// TIA Portal V16 export
// export: Created 2024-06-17T16:39:12.649221Z, ExportSetting None, DisplayName Totally Integrated Automation Portal, DisplayVersion V16, DisplayName TIA Portal Version Control Interface, DisplayVersion V16, DisplayName TIA Portal Openness, DisplayVersion V16, DisplayName STEP 7 Professional, DisplayVersion V16, DisplayName STEP 7 Safety, DisplayVersion V16, DisplayName WinCC Advanced, DisplayVersion V16
FUNCTION_BLOCK "0105_FB Robô ABB"   // FB105, LAD
TITLE = Assinatura
{ S7_Optimized_Access := 'FALSE' }
AUTHOR : Axis_Solutions
// Autor           : Pedro Mello
// E-mail         : pedro.mello@axissolutions.com.br
// Empresa    : Axis Solutions
// Site             : www.axissolutions.com.br
//                     
// Data de criação : 11.06.2024
// Função                : Gestão de robo ABB
// Comentário        : FB Standard para gestão de robo ABB
// Autor          : Pedro Mello, 
// E-mail         : Pedroeamello@hotmail.com
// Empresa        : PDR AUTOMATION
// Site           : 
//                     
// Data de criação: 01.11.2018
// Função         : FB Standard para gestão de robo ABB
// Comentário     :
// stored: AutoNumber false, SetENOAutomatically false
   VAR_INPUT
      "RB.Do_PLC.Di" : "Axis.RB.Do_PLC.Di";   // Range de Inputs do Robo
      Safety : "Axis.Safety";   // Emergencias
      IHM : "Axis.SeleçãoPainel";   // Sinais Vindos da IHM
   END_VAR
   VAR_OUTPUT
      "RB.Di_PLC.Do" : "Axis.RB.Di_PLC.Do";
   END_VAR
   VAR
      RB_Memórias { S7_SetPoint := 'True'} : "Axis.RB_Memórias";
      Start_Ciclo1 { S7_SetPoint := 'True'} : TON_TIME;   // Delay Start Ciclo
   END_VAR
   VAR_TEMP
      i : Int;
      SAVE_AR1 : DWord;
      SAVE_AR2 : DWord;
   END_VAR
   VAR CONSTANT
      False : Bool;   // Memória sempre 0
      True : Bool := True;   // Memória sempre 1
      Inicio : Int := 1;
      Fim : Int := 32;
   END_VAR
   VAR_TEMP   // added for the SCL form of the ladder/FBD networks
      _w1 : Bool;
      _w2 : Bool;
   END_VAR
BEGIN

NETWORK
TITLE = Salva Registros
      TAR1  #SAVE_AR1;
      TAR2  #SAVE_AR2;

REGION Network 2: ########## Bits de Utilidade ##########
END_REGION

REGION Network 3: ######## Automatico Sem Falhas ########
END_REGION

REGION Network 4: Delay Start Ciclo
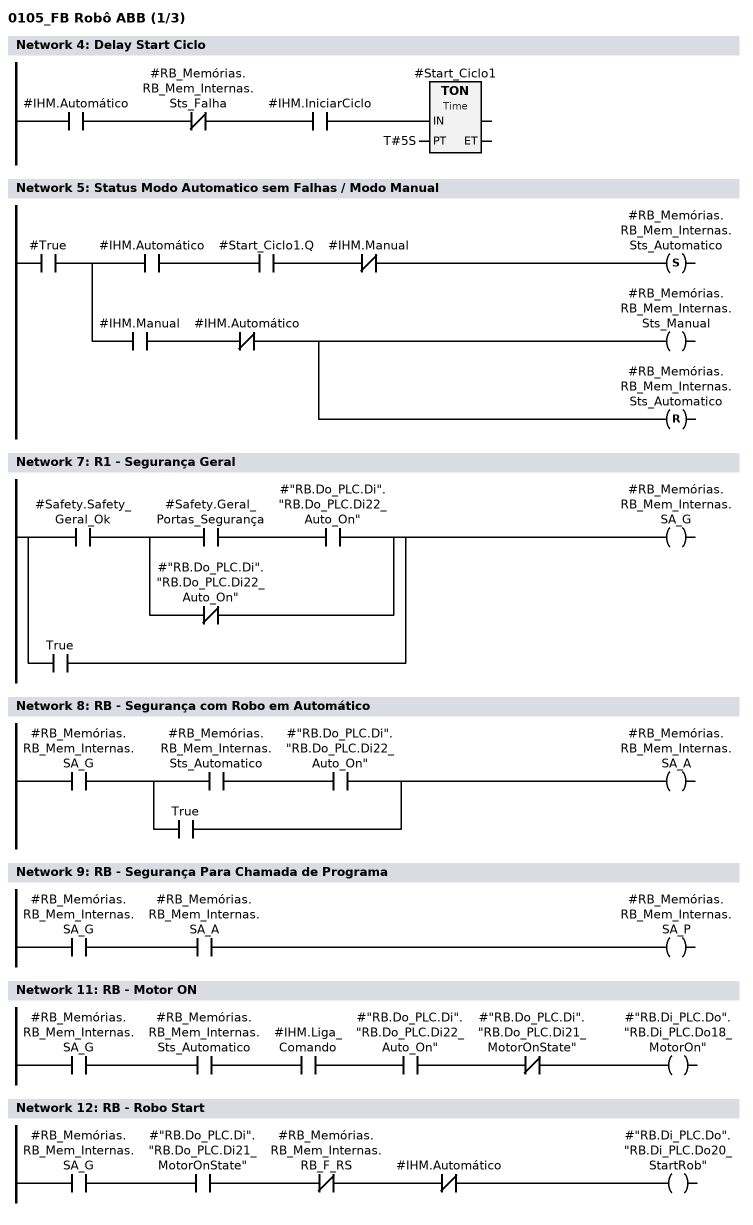
   RUNG wire#powerrail
      Contact( #IHM.Automático )
      I_Contact( #RB_Memórias.RB_Mem_Internas.Sts_Falha )
      Contact( #IHM.IniciarCiclo )
      { S7_Templates := "time_type := Time" } #Start_Ciclo1.TON(pt := T#5S, et =>)
   END_RUNG
   // the same network as SCL:
   #Start_Ciclo1(IN := #IHM.Automático AND NOT #RB_Memórias.RB_Mem_Internas.Sts_Falha AND #IHM.IniciarCiclo,   // TON
                 PT := T#5S);
END_REGION

REGION Network 5: Status Modo Automatico sem Falhas / Modo Manual
   RUNG wire#powerrail
      Contact( #True )
      wire#w1
      Contact( #IHM.Automático )
      Contact( #Start_Ciclo1.Q )
      I_Contact( #IHM.Manual )
      S_Coil( #RB_Memórias.RB_Mem_Internas.Sts_Automatico )
   END_RUNG
   RUNG wire#w1
      Contact( #IHM.Manual )
      I_Contact( #IHM.Automático )
      wire#w2
      Coil( #RB_Memórias.RB_Mem_Internas.Sts_Manual )
   END_RUNG
   RUNG wire#w2
      R_Coil( #RB_Memórias.RB_Mem_Internas.Sts_Automatico )
   END_RUNG
   // the same network as SCL:
   IF #True AND #IHM.Automático AND #Start_Ciclo1.Q AND NOT #IHM.Manual THEN
       #RB_Memórias.RB_Mem_Internas.Sts_Automatico := TRUE;
   END_IF;
   #RB_Memórias.RB_Mem_Internas.Sts_Manual := #True AND #IHM.Manual AND NOT #IHM.Automático;
   IF #RB_Memórias.RB_Mem_Internas.Sts_Manual THEN
       #RB_Memórias.RB_Mem_Internas.Sts_Automatico := FALSE;
   END_IF;
END_REGION

REGION Network 6: ########## Seguranças ##########
END_REGION

REGION Network 7: R1 - Segurança Geral
   RUNG wire#powerrail
      Contact( #Safety.Safety_Geral_Ok )
      wire#w1
      Contact( #Safety.Geral_Portas_Segurança )
      Contact( #"RB.Do_PLC.Di"."RB.Do_PLC.Di22_Auto_On" )
      wire#w2
      Coil( #RB_Memórias.RB_Mem_Internas.SA_G )
   END_RUNG
   RUNG wire#w1
      I_Contact( #"RB.Do_PLC.Di"."RB.Do_PLC.Di22_Auto_On" )
   END_RUNG wire#w2
   RUNG wire#powerrail
      Contact( True )
   END_RUNG wire#w2
   // the same network as SCL:
   #RB_Memórias.RB_Mem_Internas.SA_G := (#Safety.Safety_Geral_Ok AND ((#Safety.Geral_Portas_Segurança AND #"RB.Do_PLC.Di"."RB.Do_PLC.Di22_Auto_On") OR NOT #"RB.Do_PLC.Di"."RB.Do_PLC.Di22_Auto_On")) OR True;
END_REGION

REGION Network 8: RB - Segurança com Robo em Automático
   RUNG wire#powerrail
      Contact( #RB_Memórias.RB_Mem_Internas.SA_G )
      wire#w1
      Contact( #RB_Memórias.RB_Mem_Internas.Sts_Automatico )
      Contact( #"RB.Do_PLC.Di"."RB.Do_PLC.Di22_Auto_On" )
      wire#w2
      Coil( #RB_Memórias.RB_Mem_Internas.SA_A )
   END_RUNG
   RUNG wire#w1
      Contact( True )
   END_RUNG wire#w2
   // the same network as SCL:
   #RB_Memórias.RB_Mem_Internas.SA_A := #RB_Memórias.RB_Mem_Internas.SA_G AND ((#RB_Memórias.RB_Mem_Internas.Sts_Automatico AND #"RB.Do_PLC.Di"."RB.Do_PLC.Di22_Auto_On") OR True);
END_REGION

REGION Network 9: RB - Segurança Para Chamada de Programa
   RUNG wire#powerrail
      Contact( #RB_Memórias.RB_Mem_Internas.SA_G )
      Contact( #RB_Memórias.RB_Mem_Internas.SA_A )
      Coil( #RB_Memórias.RB_Mem_Internas.SA_P )
   END_RUNG
   // the same network as SCL:
   #RB_Memórias.RB_Mem_Internas.SA_P := #RB_Memórias.RB_Mem_Internas.SA_G AND #RB_Memórias.RB_Mem_Internas.SA_A;
END_REGION

REGION Network 10: ##################################
END_REGION

REGION Network 11: RB - Motor ON
   RUNG wire#powerrail
      Contact( #RB_Memórias.RB_Mem_Internas.SA_G )
      Contact( #RB_Memórias.RB_Mem_Internas.Sts_Automatico )
      Contact( #IHM.Liga_Comando )
      Contact( #"RB.Do_PLC.Di"."RB.Do_PLC.Di22_Auto_On" )
      I_Contact( #"RB.Do_PLC.Di"."RB.Do_PLC.Di21_MotorOnState" )
      Coil( #"RB.Di_PLC.Do"."RB.Di_PLC.Do18_MotorOn" )
   END_RUNG
   // the same network as SCL:
   #"RB.Di_PLC.Do"."RB.Di_PLC.Do18_MotorOn" := #RB_Memórias.RB_Mem_Internas.SA_G AND #RB_Memórias.RB_Mem_Internas.Sts_Automatico AND #IHM.Liga_Comando AND #"RB.Do_PLC.Di"."RB.Do_PLC.Di22_Auto_On" AND NOT #"RB.Do_PLC.Di"."RB.Do_PLC.Di21_MotorOnState";
END_REGION

REGION Network 12: RB - Robo Start
   RUNG wire#powerrail
      Contact( #RB_Memórias.RB_Mem_Internas.SA_G )
      Contact( #"RB.Do_PLC.Di"."RB.Do_PLC.Di21_MotorOnState" )
      I_Contact( #RB_Memórias.RB_Mem_Internas.RB_F_RS )
      I_Contact( #IHM.Automático )
      Coil( #"RB.Di_PLC.Do"."RB.Di_PLC.Do20_StartRob" )
   END_RUNG
   // the same network as SCL:
   #"RB.Di_PLC.Do"."RB.Di_PLC.Do20_StartRob" := #RB_Memórias.RB_Mem_Internas.SA_G AND #"RB.Do_PLC.Di"."RB.Do_PLC.Di21_MotorOnState" AND NOT #RB_Memórias.RB_Mem_Internas.RB_F_RS AND NOT #IHM.Automático;
END_REGION

REGION Network 13: RB - Memoria Robo Start
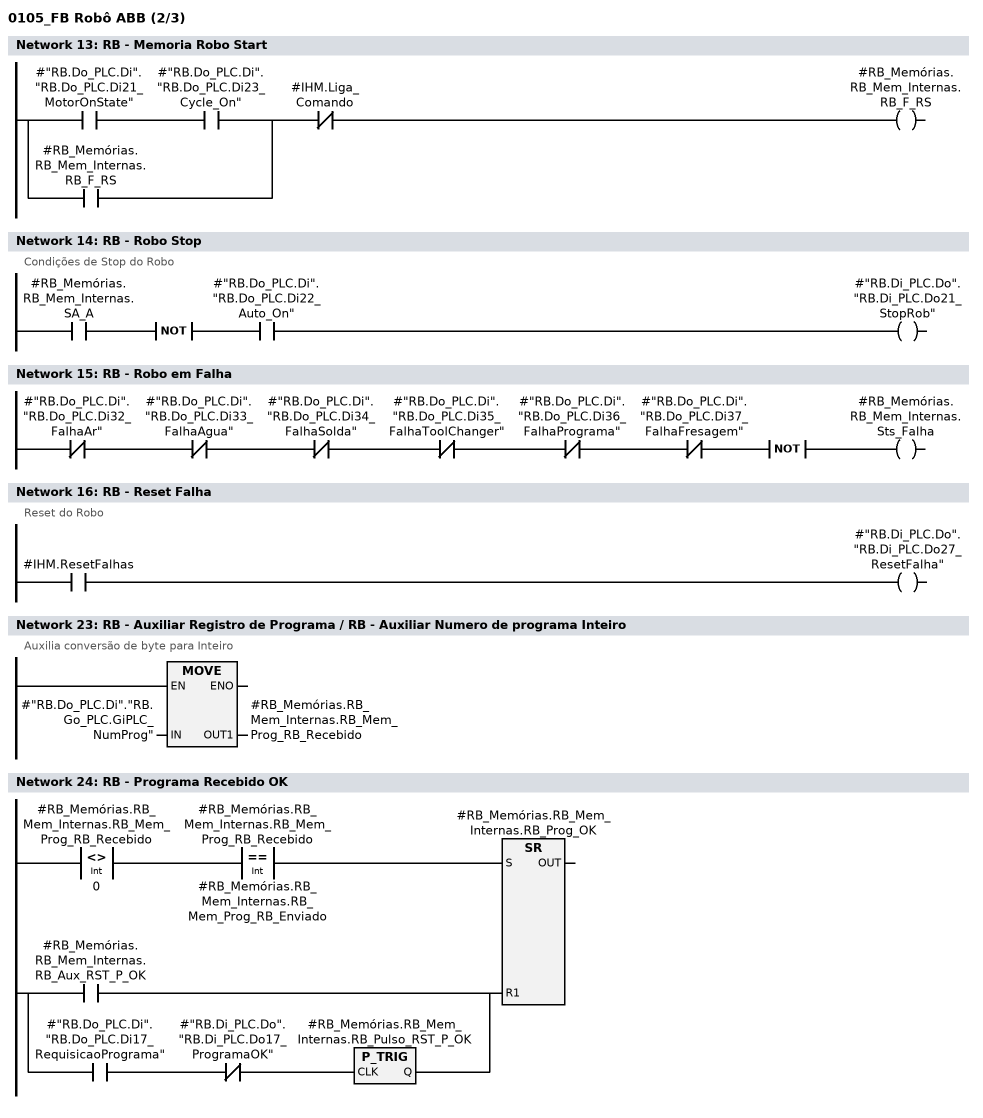
   RUNG wire#powerrail
      Contact( #"RB.Do_PLC.Di"."RB.Do_PLC.Di21_MotorOnState" )
      Contact( #"RB.Do_PLC.Di"."RB.Do_PLC.Di23_Cycle_On" )
      wire#w1
      I_Contact( #IHM.Liga_Comando )
      Coil( #RB_Memórias.RB_Mem_Internas.RB_F_RS )
   END_RUNG
   RUNG wire#powerrail
      Contact( #RB_Memórias.RB_Mem_Internas.RB_F_RS )
   END_RUNG wire#w1
   // the same network as SCL:
   #RB_Memórias.RB_Mem_Internas.RB_F_RS := ((#"RB.Do_PLC.Di"."RB.Do_PLC.Di21_MotorOnState" AND #"RB.Do_PLC.Di"."RB.Do_PLC.Di23_Cycle_On") OR #RB_Memórias.RB_Mem_Internas.RB_F_RS) AND NOT #IHM.Liga_Comando;
END_REGION

REGION Network 14: RB - Robo Stop
   // Condições de Stop do Robo
   RUNG wire#powerrail
      Contact( #RB_Memórias.RB_Mem_Internas.SA_A )
      Not()
      Contact( #"RB.Do_PLC.Di"."RB.Do_PLC.Di22_Auto_On" )
      Coil( #"RB.Di_PLC.Do"."RB.Di_PLC.Do21_StopRob" )
   END_RUNG
   // the same network as SCL:
   #"RB.Di_PLC.Do"."RB.Di_PLC.Do21_StopRob" := NOT #RB_Memórias.RB_Mem_Internas.SA_A AND #"RB.Do_PLC.Di"."RB.Do_PLC.Di22_Auto_On";
END_REGION

REGION Network 15: RB - Robo em Falha
   RUNG wire#powerrail
      I_Contact( #"RB.Do_PLC.Di"."RB.Do_PLC.Di32_FalhaAr" )
      I_Contact( #"RB.Do_PLC.Di"."RB.Do_PLC.Di33_FalhaAgua" )
      I_Contact( #"RB.Do_PLC.Di"."RB.Do_PLC.Di34_FalhaSolda" )
      I_Contact( #"RB.Do_PLC.Di"."RB.Do_PLC.Di35_FalhaToolChanger" )
      I_Contact( #"RB.Do_PLC.Di"."RB.Do_PLC.Di36_FalhaPrograma" )
      I_Contact( #"RB.Do_PLC.Di"."RB.Do_PLC.Di37_FalhaFresagem" )
      Not()
      Coil( #RB_Memórias.RB_Mem_Internas.Sts_Falha )
   END_RUNG
   // the same network as SCL:
   #RB_Memórias.RB_Mem_Internas.Sts_Falha := NOT (NOT #"RB.Do_PLC.Di"."RB.Do_PLC.Di32_FalhaAr" AND NOT #"RB.Do_PLC.Di"."RB.Do_PLC.Di33_FalhaAgua" AND NOT #"RB.Do_PLC.Di"."RB.Do_PLC.Di34_FalhaSolda" AND NOT #"RB.Do_PLC.Di"."RB.Do_PLC.Di35_FalhaToolChanger" AND NOT #"RB.Do_PLC.Di"."RB.Do_PLC.Di36_FalhaPrograma" AND NOT #"RB.Do_PLC.Di"."RB.Do_PLC.Di37_FalhaFresagem");
END_REGION

REGION Network 16: RB - Reset Falha
   // Reset do Robo
   RUNG wire#powerrail
      Contact( #IHM.ResetFalhas )
      Coil( #"RB.Di_PLC.Do"."RB.Di_PLC.Do27_ResetFalha" )
   END_RUNG
   // the same network as SCL:
   #"RB.Di_PLC.Do"."RB.Di_PLC.Do27_ResetFalha" := #IHM.ResetFalhas;
END_REGION

REGION Network 17: ########## Chamadas de Programa ##########
END_REGION

REGION Network 18 (SCL): Gerrenciamento de Programas

   //Envia Valor de Programa
   FOR #i := #Inicio TO #Fim DO
       IF  #RB_Memórias.RB_Mem_Internas.SA_P AND #"RB.Do_PLC.Di"."RB.Do_PLC.Di22_Auto_On" AND
           #"RB.Do_PLC.Di"."RB.Do_PLC.Di17_RequisicaoPrograma" AND #RB_Memórias.RB_Mem_Externas.RB_Auxiliar_de_Programa[#i] = TRUE THEN
           #"RB.Di_PLC.Do"."RB.Gi_PLC.Go_NumProg" := #i;
           #RB_Memórias.RB_Mem_Internas.RB_Mem_Prog_RB_Enviado := #i;
       END_IF;
   END_FOR;
END_REGION

REGION Network 19 (SCL): Autorização de Trabalho
   //Autorização de Trabalho_1
   IF #"RB.Do_PLC.Di"."RB.Do_PLC.Di56_AreaLivreTrab_1" AND #RB_Memórias.RB_Mem_Externas."RB_Aux_Aut.Trabalho"[1] THEN #"RB.Di_PLC.Do"."RB.Di_PLC.Do56_Aut.Trabalho_1" := TRUE;
   END_IF;
   //Autorização de Trabalho_2
   IF #"RB.Do_PLC.Di"."RB.Do_PLC.Di57_AreaLivreTrab_2" AND #RB_Memórias.RB_Mem_Externas."RB_Aux_Aut.Trabalho"[2] THEN #"RB.Di_PLC.Do"."RB.Di_PLC.Do57_Aut.Trabalho_2" := TRUE;
   END_IF;
   //Autorização de Trabalho_3
   IF #"RB.Do_PLC.Di"."RB.Do_PLC.Di58_AreaLivreTrab_3" AND #RB_Memórias.RB_Mem_Externas."RB_Aux_Aut.Trabalho"[3] THEN #"RB.Di_PLC.Do"."RB.Di_PLC.Do58_Aut.Trabalho_3" := TRUE;
   END_IF;
   //Autorização de Trabalho_4
   IF #"RB.Do_PLC.Di"."RB.Do_PLC.Di59_AreaLivreTrab_4" AND #RB_Memórias.RB_Mem_Externas."RB_Aux_Aut.Trabalho"[4] THEN #"RB.Di_PLC.Do"."RB.Di_PLC.Do59_Aut.Trabalho_4" := TRUE;
   END_IF;
   //Autorização de Trabalho_5
   IF #"RB.Do_PLC.Di"."RB.Do_PLC.Di60_AreaLivreTrab_5" AND #RB_Memórias.RB_Mem_Externas."RB_Aux_Aut.Trabalho"[5] THEN #"RB.Di_PLC.Do"."RB.Di_PLC.Do60_Aut.Trabalho_5" := TRUE;
   END_IF;
   //Autorização de Trabalho_6
   IF #"RB.Do_PLC.Di"."RB.Do_PLC.Di61_AreaLivreTrab_6" AND #RB_Memórias.RB_Mem_Externas."RB_Aux_Aut.Trabalho"[6] THEN #"RB.Di_PLC.Do"."RB.Di_PLC.Do61_Aut.Trabalho_6" := TRUE;
   END_IF;
   //Autorização de Trabalho_7
   IF #"RB.Do_PLC.Di"."RB.Do_PLC.Di62_AreaLivreTrab_7" AND #RB_Memórias.RB_Mem_Externas."RB_Aux_Aut.Trabalho"[7] THEN #"RB.Di_PLC.Do"."RB.Di_PLC.Do62_Aut.Trabalho_7" := TRUE;
   END_IF;
   //Autorização de Trabalho_8
   IF #"RB.Do_PLC.Di"."RB.Do_PLC.Di63_AreaLivreTrab_8" AND #RB_Memórias.RB_Mem_Externas."RB_Aux_Aut.Trabalho"[8] THEN #"RB.Di_PLC.Do"."RB.Di_PLC.Do63_Aut.Trabalho_8" := TRUE;
   END_IF;
   //Autorização de Trabalho_9
   IF #"RB.Do_PLC.Di"."RB.Do_PLC.Di64_AreaLivreTrab_9" AND #RB_Memórias.RB_Mem_Externas."RB_Aux_Aut.Trabalho"[9] THEN #"RB.Di_PLC.Do"."RB.Di_PLC.Do64_Aut.Trabalho_9" := TRUE;
   END_IF;
   //Autorização de Trabalho_10
   IF #"RB.Do_PLC.Di"."RB.Do_PLC.Di65_AreaLivreTrab_10" AND #RB_Memórias.RB_Mem_Externas."RB_Aux_Aut.Trabalho"[10] THEN #"RB.Di_PLC.Do"."RB.Di_PLC.Do65_Aut.Trabalho_10" := TRUE;
   END_IF;
   //Autorização de Trabalho_11
   IF #"RB.Do_PLC.Di"."RB.Do_PLC.Di66_AreaLivreTrab_11" AND #RB_Memórias.RB_Mem_Externas."RB_Aux_Aut.Trabalho"[11] THEN #"RB.Di_PLC.Do"."RB.Di_PLC.Do66_Aut.Trabalho_11" := TRUE;
   END_IF;
   //Autorização de Trabalho_12
   IF #"RB.Do_PLC.Di"."RB.Do_PLC.Di67_AreaLivreTrab_12" AND #RB_Memórias.RB_Mem_Externas."RB_Aux_Aut.Trabalho"[12] THEN #"RB.Di_PLC.Do"."RB.Di_PLC.Do67_Aut.Trabalho_12" := TRUE;
   END_IF;
   //Autorização de Trabalho_13
   IF #"RB.Do_PLC.Di"."RB.Do_PLC.Di68_AreaLivreTrab_13" AND #RB_Memórias.RB_Mem_Externas."RB_Aux_Aut.Trabalho"[13] THEN #"RB.Di_PLC.Do"."RB.Di_PLC.Do68_Aut.Trabalho_13" := TRUE;
   END_IF;
   //Autorização de Trabalho_14
   IF #"RB.Do_PLC.Di"."RB.Do_PLC.Di69_AreaLivreTrab_14" AND #RB_Memórias.RB_Mem_Externas."RB_Aux_Aut.Trabalho"[14] THEN #"RB.Di_PLC.Do"."RB.Di_PLC.Do69_Aut.Trabalho_14" := TRUE;
   END_IF;
   //Autorização de Trabalho_15
   IF #"RB.Do_PLC.Di"."RB.Do_PLC.Di70_AreaLivreTrab_15" AND #RB_Memórias.RB_Mem_Externas."RB_Aux_Aut.Trabalho"[15] THEN #"RB.Di_PLC.Do"."RB.Di_PLC.Do70_Aut.Trabalho_15" := TRUE;
   END_IF;
   //Autorização de Trabalho_16
   IF #"RB.Do_PLC.Di"."RB.Do_PLC.Di71_AreaLivreTrab_16" AND #RB_Memórias.RB_Mem_Externas."RB_Aux_Aut.Trabalho"[16] THEN #"RB.Di_PLC.Do"."RB.Di_PLC.Do71_Aut.Trabalho_16" := TRUE;
   END_IF;
   //Autorização de Trabalho_17
   IF #"RB.Do_PLC.Di"."RB.Do_PLC.Di72_AreaLivreTrab_17" AND #RB_Memórias.RB_Mem_Externas."RB_Aux_Aut.Trabalho"[17] THEN #"RB.Di_PLC.Do"."RB.Di_PLC.Do72_Aut.Trabalho_17" := TRUE;
   END_IF;
   //Autorização de Trabalho_18
   IF #"RB.Do_PLC.Di"."RB.Do_PLC.Di73_AreaLivreTrab_18" AND #RB_Memórias.RB_Mem_Externas."RB_Aux_Aut.Trabalho"[18] THEN #"RB.Di_PLC.Do"."RB.Di_PLC.Do73_Aut.Trabalho_18" := TRUE;
   END_IF;
   //Autorização de Trabalho_19
   IF #"RB.Do_PLC.Di"."RB.Do_PLC.Di74_AreaLivreTrab_19" AND #RB_Memórias.RB_Mem_Externas."RB_Aux_Aut.Trabalho"[19] THEN #"RB.Di_PLC.Do"."RB.Di_PLC.Do74_Aut.Trabalho_19" := TRUE;
   END_IF;
   //Autorização de Trabalho_20
   IF #"RB.Do_PLC.Di"."RB.Do_PLC.Di75_AreaLivreTrab_20" AND #RB_Memórias.RB_Mem_Externas."RB_Aux_Aut.Trabalho"[20] THEN #"RB.Di_PLC.Do"."RB.Di_PLC.Do75_Aut.Trabalho_20" := TRUE;
   END_IF;
   //Autorização de Trabalho_21
   IF #"RB.Do_PLC.Di"."RB.Do_PLC.Di76_AreaLivreTrab_21" AND #RB_Memórias.RB_Mem_Externas."RB_Aux_Aut.Trabalho"[21] THEN #"RB.Di_PLC.Do"."RB.Di_PLC.Do76_Aut.Trabalho_21" := TRUE;
   END_IF;
   //Autorização de Trabalho_22
   IF #"RB.Do_PLC.Di"."RB.Do_PLC.Di77_AreaLivreTrab_22" AND #RB_Memórias.RB_Mem_Externas."RB_Aux_Aut.Trabalho"[22] THEN #"RB.Di_PLC.Do"."RB.Di_PLC.Do77_Aut.Trabalho_22" := TRUE;
   END_IF;
   //Autorização de Trabalho_23
   IF #"RB.Do_PLC.Di"."RB.Do_PLC.Di78_AreaLivreTrab_23" AND #RB_Memórias.RB_Mem_Externas."RB_Aux_Aut.Trabalho"[23] THEN #"RB.Di_PLC.Do"."RB.Di_PLC.Do78_Aut.Trabalho_23" := TRUE;
   END_IF;
   //Autorização de Trabalho_24
   IF #"RB.Do_PLC.Di"."RB.Do_PLC.Di79_AreaLivreTrab_24" AND #RB_Memórias.RB_Mem_Externas."RB_Aux_Aut.Trabalho"[24] THEN #"RB.Di_PLC.Do"."RB.Di_PLC.Do79_Aut.Trabalho_24" := TRUE;
   END_IF;
   //Autorização de Trabalho_25
   IF #"RB.Do_PLC.Di"."RB.Do_PLC.Di80_AreaLivreTrab_25" AND #RB_Memórias.RB_Mem_Externas."RB_Aux_Aut.Trabalho"[25] THEN #"RB.Di_PLC.Do"."RB.Di_PLC.Do80_Aut.Trabalho_25" := TRUE;
   END_IF;
   //Autorização de Trabalho_26
   IF #"RB.Do_PLC.Di"."RB.Do_PLC.Di81_AreaLivreTrab_26" AND #RB_Memórias.RB_Mem_Externas."RB_Aux_Aut.Trabalho"[26] THEN #"RB.Di_PLC.Do"."RB.Di_PLC.Do81_Aut.Trabalho_26" := TRUE;
   END_IF;
   //Autorização de Trabalho_27
   IF #"RB.Do_PLC.Di"."RB.Do_PLC.Di82_AreaLivreTrab_27" AND #RB_Memórias.RB_Mem_Externas."RB_Aux_Aut.Trabalho"[27] THEN #"RB.Di_PLC.Do"."RB.Di_PLC.Do82_Aut.Trabalho_27" := TRUE;
   END_IF;
   //Autorização de Trabalho_28
   IF #"RB.Do_PLC.Di"."RB.Do_PLC.Di83_AreaLivreTrab_28" AND #RB_Memórias.RB_Mem_Externas."RB_Aux_Aut.Trabalho"[28] THEN #"RB.Di_PLC.Do"."RB.Di_PLC.Do83_Aut.Trabalho_28" := TRUE;
   END_IF;
   //Autorização de Trabalho_29
   IF #"RB.Do_PLC.Di"."RB.Do_PLC.Di84_AreaLivreTrab_29" AND #RB_Memórias.RB_Mem_Externas."RB_Aux_Aut.Trabalho"[29] THEN #"RB.Di_PLC.Do"."RB.Di_PLC.Do84_Aut.Trabalho_29" := TRUE;
   END_IF;
   //Autorização de Trabalho_30
   IF #"RB.Do_PLC.Di"."RB.Do_PLC.Di85_AreaLivreTrab_30" AND #RB_Memórias.RB_Mem_Externas."RB_Aux_Aut.Trabalho"[30] THEN #"RB.Di_PLC.Do"."RB.Di_PLC.Do85_Aut.Trabalho_30" := TRUE;
   END_IF;
   //Autorização de Trabalho_31
   IF #"RB.Do_PLC.Di"."RB.Do_PLC.Di86_AreaLivreTrab_31" AND #RB_Memórias.RB_Mem_Externas."RB_Aux_Aut.Trabalho"[31] THEN #"RB.Di_PLC.Do"."RB.Di_PLC.Do86_Aut.Trabalho_31" := TRUE;
   END_IF;
   //Autorização de Trabalho_32
   IF #"RB.Do_PLC.Di"."RB.Do_PLC.Di87_AreaLivreTrab_32" AND #RB_Memórias.RB_Mem_Externas."RB_Aux_Aut.Trabalho"[32] THEN #"RB.Di_PLC.Do"."RB.Di_PLC.Do87_Aut.Trabalho_32" := TRUE;
   END_IF;
END_REGION

REGION Network 20 (SCL): Autorização de Intertravamento
   //Autorização de Intertravamento_1
   IF #"RB.Do_PLC.Di"."RB.Do_PLC.Di88_Intertravamento_1" AND #RB_Memórias.RB_Mem_Externas."RB_Aux_Aut.Intertravamento"[1] THEN #"RB.Di_PLC.Do"."RB.Di_PLC.Do88_Aut.Intertravamento_1" := TRUE;
   END_IF;
   //Autorização de Intertravamento_2
   IF #"RB.Do_PLC.Di"."RB.Do_PLC.Di89_Intertravamento_2" AND #RB_Memórias.RB_Mem_Externas."RB_Aux_Aut.Intertravamento"[2] THEN #"RB.Di_PLC.Do"."RB.Di_PLC.Do89_Aut.Intertravamento_2" := TRUE;
   END_IF;
   //Autorização de Intertravamento_3
   IF #"RB.Do_PLC.Di"."RB.Do_PLC.Di90_Intertravamento_3" AND #RB_Memórias.RB_Mem_Externas."RB_Aux_Aut.Intertravamento"[3] THEN #"RB.Di_PLC.Do"."RB.Di_PLC.Do90_Aut.Intertravamento_3" := TRUE;
   END_IF;
   //Autorização de Intertravamento_4
   IF #"RB.Do_PLC.Di"."RB.Do_PLC.Di91_Intertravamento_4" AND #RB_Memórias.RB_Mem_Externas."RB_Aux_Aut.Intertravamento"[4] THEN #"RB.Di_PLC.Do"."RB.Di_PLC.Do91_Aut.Intertravamento_4" := TRUE;
   END_IF;
   //Autorização de Intertravamento_5
   IF #"RB.Do_PLC.Di"."RB.Do_PLC.Di92_Intertravamento_5" AND #RB_Memórias.RB_Mem_Externas."RB_Aux_Aut.Intertravamento"[5] THEN #"RB.Di_PLC.Do"."RB.Di_PLC.Do92_Aut.Intertravamento_5" := TRUE;
   END_IF;
   //Autorização de Intertravamento_6
   IF #"RB.Do_PLC.Di"."RB.Do_PLC.Di93_Intertravamento_6" AND #RB_Memórias.RB_Mem_Externas."RB_Aux_Aut.Intertravamento"[6] THEN #"RB.Di_PLC.Do"."RB.Di_PLC.Do93_Aut.Intertravamento_6" := TRUE;
   END_IF;
   //Autorização de Intertravamento_7
   IF #"RB.Do_PLC.Di"."RB.Do_PLC.Di94_Intertravamento_7" AND #RB_Memórias.RB_Mem_Externas."RB_Aux_Aut.Intertravamento"[7] THEN #"RB.Di_PLC.Do"."RB.Di_PLC.Do94_Aut.Intertravamento_7" := TRUE;
   END_IF;
   //Autorização de Intertravamento_8
   IF #"RB.Do_PLC.Di"."RB.Do_PLC.Di95_Intertravamento_8" AND #RB_Memórias.RB_Mem_Externas."RB_Aux_Aut.Intertravamento"[8] THEN #"RB.Di_PLC.Do"."RB.Di_PLC.Do95_Aut.Intertravamento_8" := TRUE;
   END_IF;
   //Autorização de Intertravamento_9
   IF #"RB.Do_PLC.Di"."RB.Do_PLC.Di96_Intertravamento_9" AND #RB_Memórias.RB_Mem_Externas."RB_Aux_Aut.Intertravamento"[9] THEN #"RB.Di_PLC.Do"."RB.Di_PLC.Do96_Aut.Intertravamento_9" := TRUE;
   END_IF;
   //Autorização de Intertravamento_10
   IF #"RB.Do_PLC.Di"."RB.Do_PLC.Di97_Intertravamento_10" AND #RB_Memórias.RB_Mem_Externas."RB_Aux_Aut.Intertravamento"[10] THEN #"RB.Di_PLC.Do"."RB.Di_PLC.Do97_Aut.Intertravamento_10" := TRUE;
   END_IF;
   //Autorização de Intertravamento_11
   IF #"RB.Do_PLC.Di"."RB.Do_PLC.Di98_Intertravamento_11" AND #RB_Memórias.RB_Mem_Externas."RB_Aux_Aut.Intertravamento"[11] THEN #"RB.Di_PLC.Do"."RB.Di_PLC.Do98_Aut.Intertravamento_11" := TRUE;
   END_IF;
   //Autorização de Intertravamento_12
   IF #"RB.Do_PLC.Di"."RB.Do_PLC.Di99_Intertravamento_12" AND #RB_Memórias.RB_Mem_Externas."RB_Aux_Aut.Intertravamento"[12] THEN #"RB.Di_PLC.Do"."RB.Di_PLC.Do99_Aut.Intertravamento_12" := TRUE;
   END_IF;
   //Autorização de Intertravamento_13
   IF #"RB.Do_PLC.Di"."RB.Do_PLC.Di100_Intertravamento_13" AND #RB_Memórias.RB_Mem_Externas."RB_Aux_Aut.Intertravamento"[13] THEN #"RB.Di_PLC.Do"."RB.Di_PLC.Do100_Aut.Intertravamento_13" := TRUE;
   END_IF;
   //Autorização de Intertravamento_14
   IF #"RB.Do_PLC.Di"."RB.Do_PLC.Di101_Intertravamento_14" AND #RB_Memórias.RB_Mem_Externas."RB_Aux_Aut.Intertravamento"[14] THEN #"RB.Di_PLC.Do"."RB.Di_PLC.Do101_Aut.Intertravamento_14" := TRUE;
   END_IF;
   //Autorização de Intertravamento_15
   IF #"RB.Do_PLC.Di"."RB.Do_PLC.Di102_Intertravamento_15" AND #RB_Memórias.RB_Mem_Externas."RB_Aux_Aut.Intertravamento"[15] THEN #"RB.Di_PLC.Do"."RB.Di_PLC.Do102_Aut.Intertravamento_15" := TRUE;
   END_IF;
   //Autorização de Intertravamento_16
   IF #"RB.Do_PLC.Di"."RB.Do_PLC.Di103_Intertravamento_16" AND #RB_Memórias.RB_Mem_Externas."RB_Aux_Aut.Intertravamento"[16] THEN #"RB.Di_PLC.Do"."RB.Di_PLC.Do103_Aut.Intertravamento_16" := TRUE;
   END_IF;
   //Autorização de Intertravamento_17
   IF #"RB.Do_PLC.Di"."RB.Do_PLC.Di104_Intertravamento_17" AND #RB_Memórias.RB_Mem_Externas."RB_Aux_Aut.Intertravamento"[17] THEN #"RB.Di_PLC.Do"."RB.Di_PLC.Do104_Aut.Intertravamento_17" := TRUE;
   END_IF;
   //Autorização de Intertravamento_18
   IF #"RB.Do_PLC.Di"."RB.Do_PLC.Di105_Intertravamento_18" AND #RB_Memórias.RB_Mem_Externas."RB_Aux_Aut.Intertravamento"[18] THEN #"RB.Di_PLC.Do"."RB.Di_PLC.Do105_Aut.Intertravamento_18" := TRUE;
   END_IF;
   //Autorização de Intertravamento_19
   IF #"RB.Do_PLC.Di"."RB.Do_PLC.Di106_Intertravamento_19" AND #RB_Memórias.RB_Mem_Externas."RB_Aux_Aut.Intertravamento"[19] THEN #"RB.Di_PLC.Do"."RB.Di_PLC.Do106_Aut.Intertravamento_19" := TRUE;
   END_IF;
   //Autorização de Intertravamento_20
   IF #"RB.Do_PLC.Di"."RB.Do_PLC.Di107_Intertravamento_20" AND #RB_Memórias.RB_Mem_Externas."RB_Aux_Aut.Intertravamento"[20] THEN #"RB.Di_PLC.Do"."RB.Di_PLC.Do107_Aut.Intertravamento_20" := TRUE;
   END_IF;
   //Autorização de Intertravamento_21
   IF #"RB.Do_PLC.Di"."RB.Do_PLC.Di108_Intertravamento_21" AND #RB_Memórias.RB_Mem_Externas."RB_Aux_Aut.Intertravamento"[21] THEN #"RB.Di_PLC.Do"."RB.Di_PLC.Do108_Aut.Intertravamento_21" := TRUE;
   END_IF;
   //Autorização de Intertravamento_22
   IF #"RB.Do_PLC.Di"."RB.Do_PLC.Di109_Intertravamento_22" AND #RB_Memórias.RB_Mem_Externas."RB_Aux_Aut.Intertravamento"[22] THEN #"RB.Di_PLC.Do"."RB.Di_PLC.Do109_Aut.Intertravamento_22" := TRUE;
   END_IF;
   //Autorização de Intertravamento_23
   IF #"RB.Do_PLC.Di"."RB.Do_PLC.Di110_Intertravamento_23" AND #RB_Memórias.RB_Mem_Externas."RB_Aux_Aut.Intertravamento"[23] THEN #"RB.Di_PLC.Do"."RB.Di_PLC.Do110_Aut.Intertravamento_23" := TRUE;
   END_IF;
   //Autorização de Intertravamento_24
   IF #"RB.Do_PLC.Di"."RB.Do_PLC.Di111_Intertravamento_24" AND #RB_Memórias.RB_Mem_Externas."RB_Aux_Aut.Intertravamento"[24] THEN #"RB.Di_PLC.Do"."RB.Di_PLC.Do111_Aut.Intertravamento_24" := TRUE;
   END_IF;
   //Autorização de Intertravamento_25
   IF #"RB.Do_PLC.Di"."RB.Do_PLC.Di112_Intertravamento_25" AND #RB_Memórias.RB_Mem_Externas."RB_Aux_Aut.Intertravamento"[25] THEN #"RB.Di_PLC.Do"."RB.Di_PLC.Do112_Aut.Intertravamento_25" := TRUE;
   END_IF;
   //Autorização de Intertravamento_26
   IF #"RB.Do_PLC.Di"."RB.Do_PLC.Di113_Intertravamento_26" AND #RB_Memórias.RB_Mem_Externas."RB_Aux_Aut.Intertravamento"[26] THEN #"RB.Di_PLC.Do"."RB.Di_PLC.Do113_Aut.Intertravamento_26" := TRUE;
   END_IF;
   //Autorização de Intertravamento_27
   IF #"RB.Do_PLC.Di"."RB.Do_PLC.Di114_Intertravamento_27" AND #RB_Memórias.RB_Mem_Externas."RB_Aux_Aut.Intertravamento"[27] THEN #"RB.Di_PLC.Do"."RB.Di_PLC.Do114_Aut.Intertravamento_27" := TRUE;
   END_IF;
   //Autorização de Intertravamento_28
   IF #"RB.Do_PLC.Di"."RB.Do_PLC.Di115_Intertravamento_28" AND #RB_Memórias.RB_Mem_Externas."RB_Aux_Aut.Intertravamento"[28] THEN #"RB.Di_PLC.Do"."RB.Di_PLC.Do115_Aut.Intertravamento_28" := TRUE;
   END_IF;
   //Autorização de Intertravamento_29
   IF #"RB.Do_PLC.Di"."RB.Do_PLC.Di116_Intertravamento_29" AND #RB_Memórias.RB_Mem_Externas."RB_Aux_Aut.Intertravamento"[29] THEN #"RB.Di_PLC.Do"."RB.Di_PLC.Do116_Aut.Intertravamento_29" := TRUE;
   END_IF;
   //Autorização de Intertravamento_30
   IF #"RB.Do_PLC.Di"."RB.Do_PLC.Di117_Intertravamento_30" AND #RB_Memórias.RB_Mem_Externas."RB_Aux_Aut.Intertravamento"[30] THEN #"RB.Di_PLC.Do"."RB.Di_PLC.Do117_Aut.Intertravamento_30" := TRUE;
   END_IF;
   //Autorização de Intertravamento_31
   IF #"RB.Do_PLC.Di"."RB.Do_PLC.Di118_Intertravamento_31" AND #RB_Memórias.RB_Mem_Externas."RB_Aux_Aut.Intertravamento"[31] THEN #"RB.Di_PLC.Do"."RB.Di_PLC.Do118_Aut.Intertravamento_31" := TRUE;
   END_IF;
   //Autorização de Intertravamento_32
   IF #"RB.Do_PLC.Di"."RB.Do_PLC.Di119_Intertravamento_32" AND #RB_Memórias.RB_Mem_Externas."RB_Aux_Aut.Intertravamento"[32] THEN #"RB.Di_PLC.Do"."RB.Di_PLC.Do119_Aut.Intertravamento_32" := TRUE;
   END_IF;
END_REGION

REGION Network 21 (SCL): Reconhece Fim de Trabalho
   //Reconhece Fim de Trabalho_1
   IF #"RB.Do_PLC.Di"."RB.Do_PLC.Di120_FimTrabalho_1" AND #RB_Memórias.RB_Mem_Externas."RB_Aux_Rec.FimTrabalho"[1] THEN #"RB.Di_PLC.Do"."RB.Di_PLC.Do120_Rec.FimTrabalho_1" := TRUE;
   END_IF;
   //Reconhece Fim de Trabalho_2
   IF #"RB.Do_PLC.Di"."RB.Do_PLC.Di121_FimTrabalho_2" AND #RB_Memórias.RB_Mem_Externas."RB_Aux_Rec.FimTrabalho"[2] THEN #"RB.Di_PLC.Do"."RB.Di_PLC.Do121_Rec.FimTrabalho_2" := TRUE;
   END_IF;
   //Reconhece Fim de Trabalho_3
   IF #"RB.Do_PLC.Di"."RB.Do_PLC.Di122_FimTrabalho_3" AND #RB_Memórias.RB_Mem_Externas."RB_Aux_Rec.FimTrabalho"[3] THEN #"RB.Di_PLC.Do"."RB.Di_PLC.Do122_Rec.FimTrabalho_3" := TRUE;
   END_IF;
   //Reconhece Fim de Trabalho_4
   IF #"RB.Do_PLC.Di"."RB.Do_PLC.Di123_FimTrabalho_4" AND #RB_Memórias.RB_Mem_Externas."RB_Aux_Rec.FimTrabalho"[4] THEN #"RB.Di_PLC.Do"."RB.Di_PLC.Do123_Rec.FimTrabalho_4" := TRUE;
   END_IF;
   //Reconhece Fim de Trabalho_5
   IF #"RB.Do_PLC.Di"."RB.Do_PLC.Di124_FimTrabalho_5" AND #RB_Memórias.RB_Mem_Externas."RB_Aux_Rec.FimTrabalho"[5] THEN #"RB.Di_PLC.Do"."RB.Di_PLC.Do124_Rec.FimTrabalho_5" := TRUE;
   END_IF;
   //Reconhece Fim de Trabalho_6
   IF #"RB.Do_PLC.Di"."RB.Do_PLC.Di125_FimTrabalho_6" AND #RB_Memórias.RB_Mem_Externas."RB_Aux_Rec.FimTrabalho"[6] THEN #"RB.Di_PLC.Do"."RB.Di_PLC.Do125_Rec.FimTrabalho_6" := TRUE;
   END_IF;
   //Reconhece Fim de Trabalho_7
   IF #"RB.Do_PLC.Di"."RB.Do_PLC.Di126_FimTrabalho_7" AND #RB_Memórias.RB_Mem_Externas."RB_Aux_Rec.FimTrabalho"[7] THEN #"RB.Di_PLC.Do"."RB.Di_PLC.Do126_Rec.FimTrabalho_7" := TRUE;
   END_IF;
   //Reconhece Fim de Trabalho_8
   IF #"RB.Do_PLC.Di"."RB.Do_PLC.Di127_FimTrabalho_8" AND #RB_Memórias.RB_Mem_Externas."RB_Aux_Rec.FimTrabalho"[8] THEN #"RB.Di_PLC.Do"."RB.Di_PLC.Do127_Rec.FimTrabalho_8" := TRUE;
   END_IF;
   //Reconhece Fim de Trabalho_9
   IF #"RB.Do_PLC.Di"."RB.Do_PLC.Di128_FimTrabalho_9" AND #RB_Memórias.RB_Mem_Externas."RB_Aux_Rec.FimTrabalho"[9] THEN #"RB.Di_PLC.Do"."RB.Di_PLC.Do128_Rec.FimTrabalho_9" := TRUE;
   END_IF;
   //Reconhece Fim de Trabalho_10
   IF #"RB.Do_PLC.Di"."RB.Do_PLC.Di129_FimTrabalho_10" AND #RB_Memórias.RB_Mem_Externas."RB_Aux_Rec.FimTrabalho"[10] THEN #"RB.Di_PLC.Do"."RB.Di_PLC.Do129_Rec.FimTrabalho_10" := TRUE;
   END_IF;
   //Reconhece Fim de Trabalho_11
   IF #"RB.Do_PLC.Di"."RB.Do_PLC.Di130_FimTrabalho_11" AND #RB_Memórias.RB_Mem_Externas."RB_Aux_Rec.FimTrabalho"[11] THEN #"RB.Di_PLC.Do"."RB.Di_PLC.Do130_Rec.FimTrabalho_11" := TRUE;
   END_IF;
   //Reconhece Fim de Trabalho_12
   IF #"RB.Do_PLC.Di"."RB.Do_PLC.Di131_FimTrabalho_12" AND #RB_Memórias.RB_Mem_Externas."RB_Aux_Rec.FimTrabalho"[12] THEN #"RB.Di_PLC.Do"."RB.Di_PLC.Do131_Rec.FimTrabalho_12" := TRUE;
   END_IF;
   //Reconhece Fim de Trabalho_13
   IF #"RB.Do_PLC.Di"."RB.Do_PLC.Di132_FimTrabalho_13" AND #RB_Memórias.RB_Mem_Externas."RB_Aux_Rec.FimTrabalho"[13] THEN #"RB.Di_PLC.Do"."RB.Di_PLC.Do132_Rec.FimTrabalho_13" := TRUE;
   END_IF;
   //Reconhece Fim de Trabalho_14
   IF #"RB.Do_PLC.Di"."RB.Do_PLC.Di133_FimTrabalho_14" AND #RB_Memórias.RB_Mem_Externas."RB_Aux_Rec.FimTrabalho"[14] THEN #"RB.Di_PLC.Do"."RB.Di_PLC.Do133_Rec.FimTrabalho_14" := TRUE;
   END_IF;
   //Reconhece Fim de Trabalho_15
   IF #"RB.Do_PLC.Di"."RB.Do_PLC.Di134_FimTrabalho_15" AND #RB_Memórias.RB_Mem_Externas."RB_Aux_Rec.FimTrabalho"[15] THEN #"RB.Di_PLC.Do"."RB.Di_PLC.Do134_Rec.FimTrabalho_15" := TRUE;
   END_IF;
   //Reconhece Fim de Trabalho_16
   IF #"RB.Do_PLC.Di"."RB.Do_PLC.Di135_FimTrabalho_16" AND #RB_Memórias.RB_Mem_Externas."RB_Aux_Rec.FimTrabalho"[16] THEN #"RB.Di_PLC.Do"."RB.Di_PLC.Do135_Rec.FimTrabalho_16" := TRUE;
   END_IF;
   //Reconhece Fim de Trabalho_17
   IF #"RB.Do_PLC.Di"."RB.Do_PLC.Di136_FimTrabalho_17" AND #RB_Memórias.RB_Mem_Externas."RB_Aux_Rec.FimTrabalho"[17] THEN #"RB.Di_PLC.Do"."RB.Di_PLC.Do136_Rec.FimTrabalho_17" := TRUE;
   END_IF;
   //Reconhece Fim de Trabalho_18
   IF #"RB.Do_PLC.Di"."RB.Do_PLC.Di137_FimTrabalho_18" AND #RB_Memórias.RB_Mem_Externas."RB_Aux_Rec.FimTrabalho"[18] THEN #"RB.Di_PLC.Do"."RB.Di_PLC.Do137_Rec.FimTrabalho_18" := TRUE;
   END_IF;
   //Reconhece Fim de Trabalho_19
   IF #"RB.Do_PLC.Di"."RB.Do_PLC.Di138_FimTrabalho_19" AND #RB_Memórias.RB_Mem_Externas."RB_Aux_Rec.FimTrabalho"[19] THEN #"RB.Di_PLC.Do"."RB.Di_PLC.Do138_Rec.FimTrabalho_19" := TRUE;
   END_IF;
   //Reconhece Fim de Trabalho_20
   IF #"RB.Do_PLC.Di"."RB.Do_PLC.Di139_FimTrabalho_20" AND #RB_Memórias.RB_Mem_Externas."RB_Aux_Rec.FimTrabalho"[20] THEN #"RB.Di_PLC.Do"."RB.Di_PLC.Do139_Rec.FimTrabalho_20" := TRUE;
   END_IF;
   //Reconhece Fim de Trabalho_21
   IF #"RB.Do_PLC.Di"."RB.Do_PLC.Di140_FimTrabalho_21" AND #RB_Memórias.RB_Mem_Externas."RB_Aux_Rec.FimTrabalho"[21] THEN #"RB.Di_PLC.Do"."RB.Di_PLC.Do140_Rec.FimTrabalho_21" := TRUE;
   END_IF;
   //Reconhece Fim de Trabalho_22
   IF #"RB.Do_PLC.Di"."RB.Do_PLC.Di141_FimTrabalho_22" AND #RB_Memórias.RB_Mem_Externas."RB_Aux_Rec.FimTrabalho"[22] THEN #"RB.Di_PLC.Do"."RB.Di_PLC.Do141_Rec.FimTrabalho_22" := TRUE;
   END_IF;
   //Reconhece Fim de Trabalho_23
   IF #"RB.Do_PLC.Di"."RB.Do_PLC.Di142_FimTrabalho_23" AND #RB_Memórias.RB_Mem_Externas."RB_Aux_Rec.FimTrabalho"[23] THEN #"RB.Di_PLC.Do"."RB.Di_PLC.Do142_Rec.FimTrabalho_23" := TRUE;
   END_IF;
   //Reconhece Fim de Trabalho_24
   IF #"RB.Do_PLC.Di"."RB.Do_PLC.Di143_FimTrabalho_24" AND #RB_Memórias.RB_Mem_Externas."RB_Aux_Rec.FimTrabalho"[24] THEN #"RB.Di_PLC.Do"."RB.Di_PLC.Do143_Rec.FimTrabalho_24" := TRUE;
   END_IF;
   //Reconhece Fim de Trabalho_25
   IF #"RB.Do_PLC.Di"."RB.Do_PLC.Di144_FimTrabalho_25" AND #RB_Memórias.RB_Mem_Externas."RB_Aux_Rec.FimTrabalho"[25] THEN #"RB.Di_PLC.Do"."RB.Di_PLC.Do144_Rec.FimTrabalho_25" := TRUE;
   END_IF;
   //Reconhece Fim de Trabalho_26
   IF #"RB.Do_PLC.Di"."RB.Do_PLC.Di145_FimTrabalho_26" AND #RB_Memórias.RB_Mem_Externas."RB_Aux_Rec.FimTrabalho"[26] THEN #"RB.Di_PLC.Do"."RB.Di_PLC.Do145_Rec.FimTrabalho_26" := TRUE;
   END_IF;
   //Reconhece Fim de Trabalho_27
   IF #"RB.Do_PLC.Di"."RB.Do_PLC.Di146_FimTrabalho_27" AND #RB_Memórias.RB_Mem_Externas."RB_Aux_Rec.FimTrabalho"[27] THEN #"RB.Di_PLC.Do"."RB.Di_PLC.Do146_Rec.FimTrabalho_27" := TRUE;
   END_IF;
   //Reconhece Fim de Trabalho_28
   IF #"RB.Do_PLC.Di"."RB.Do_PLC.Di147_FimTrabalho_28" AND #RB_Memórias.RB_Mem_Externas."RB_Aux_Rec.FimTrabalho"[28] THEN #"RB.Di_PLC.Do"."RB.Di_PLC.Do147_Rec.FimTrabalho_28" := TRUE;
   END_IF;
   //Reconhece Fim de Trabalho_29
   IF #"RB.Do_PLC.Di"."RB.Do_PLC.Di148_FimTrabalho_29" AND #RB_Memórias.RB_Mem_Externas."RB_Aux_Rec.FimTrabalho"[29] THEN #"RB.Di_PLC.Do"."RB.Di_PLC.Do148_Rec.FimTrabalho_29" := TRUE;
   END_IF;
   //Reconhece Fim de Trabalho_30
   IF #"RB.Do_PLC.Di"."RB.Do_PLC.Di149_FimTrabalho_30" AND #RB_Memórias.RB_Mem_Externas."RB_Aux_Rec.FimTrabalho"[30] THEN #"RB.Di_PLC.Do"."RB.Di_PLC.Do149_Rec.FimTrabalho_30" := TRUE;
   END_IF;
   //Reconhece Fim de Trabalho_31
   IF #"RB.Do_PLC.Di"."RB.Do_PLC.Di150_FimTrabalho_31" AND #RB_Memórias.RB_Mem_Externas."RB_Aux_Rec.FimTrabalho"[31] THEN #"RB.Di_PLC.Do"."RB.Di_PLC.Do150_Rec.FimTrabalho_31" := TRUE;
   END_IF;
   //Reconhece Fim de Trabalho_32
   IF #"RB.Do_PLC.Di"."RB.Do_PLC.Di151_FimTrabalho_32" AND #RB_Memórias.RB_Mem_Externas."RB_Aux_Rec.FimTrabalho"[32] THEN #"RB.Di_PLC.Do"."RB.Di_PLC.Do151_Rec.FimTrabalho_32" := TRUE;
   END_IF;
END_REGION

REGION Network 22: ###########################################
END_REGION

REGION Network 23: RB - Auxiliar Registro de Programa / RB - Auxiliar Numero de programa Inteiro
   // Auxilia conversão de byte para Inteiro
   RUNG wire#powerrail
      { S7_GenerateENO := "TRUE" } Move(in := #"RB.Do_PLC.Di"."RB.Go_PLC.GiPLC_NumProg", out1 => #RB_Memórias.RB_Mem_Internas.RB_Mem_Prog_RB_Recebido)
   END_RUNG
   // the same network as SCL:
   #RB_Memórias.RB_Mem_Internas.RB_Mem_Prog_RB_Recebido := #"RB.Do_PLC.Di"."RB.Go_PLC.GiPLC_NumProg";
END_REGION

REGION Network 24: RB - Programa Recebido OK
   RUNG wire#powerrail
      { S7_Templates := "SrcType := Int" } NE_Contact(in1 := #RB_Memórias.RB_Mem_Internas.RB_Mem_Prog_RB_Recebido, in2 := 0)
      { S7_Templates := "SrcType := Int" } EQ_Contact(in1 := #RB_Memórias.RB_Mem_Internas.RB_Mem_Prog_RB_Recebido, in2 := #RB_Memórias.RB_Mem_Internas.RB_Mem_Prog_RB_Enviado)
      S_SR(operand := #RB_Memórias.RB_Mem_Internas.RB_Prog_OK, r1 := wire#w1)
   END_RUNG
   RUNG wire#powerrail
      Contact( #RB_Memórias.RB_Mem_Internas.RB_Aux_RST_P_OK )
   END_RUNG wire#w1
   RUNG wire#powerrail
      Contact( #"RB.Do_PLC.Di"."RB.Do_PLC.Di17_RequisicaoPrograma" )
      I_Contact( #"RB.Di_PLC.Do"."RB.Di_PLC.Do17_ProgramaOK" )
      P_Trig( #RB_Memórias.RB_Mem_Internas.RB_Pulso_RST_P_OK )
   END_RUNG wire#w1
   // the same network as SCL:
   #_w1 := #"RB.Do_PLC.Di"."RB.Do_PLC.Di17_RequisicaoPrograma" AND NOT #"RB.Di_PLC.Do"."RB.Di_PLC.Do17_ProgramaOK";
   #_w2 := #_w1 AND NOT #RB_Memórias.RB_Mem_Internas.RB_Pulso_RST_P_OK;   // rising edge
   #RB_Memórias.RB_Mem_Internas.RB_Pulso_RST_P_OK := #_w1;
   IF (#RB_Memórias.RB_Mem_Internas.RB_Mem_Prog_RB_Recebido <> 0) AND (#RB_Memórias.RB_Mem_Internas.RB_Mem_Prog_RB_Recebido = #RB_Memórias.RB_Mem_Internas.RB_Mem_Prog_RB_Enviado) THEN
       #RB_Memórias.RB_Mem_Internas.RB_Prog_OK := TRUE;   // SR flip-flop
   END_IF;
   IF #RB_Memórias.RB_Mem_Internas.RB_Aux_RST_P_OK OR #_w2 THEN
       #RB_Memórias.RB_Mem_Internas.RB_Prog_OK := FALSE;
   END_IF;
END_REGION

REGION Network 25: RB - Confirmação de Programa OK para o Robô
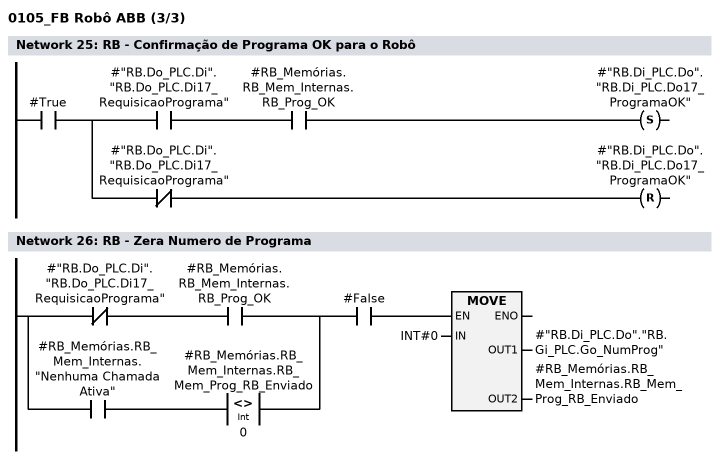
   RUNG wire#powerrail
      Contact( #True )
      wire#w1
      Contact( #"RB.Do_PLC.Di"."RB.Do_PLC.Di17_RequisicaoPrograma" )
      Contact( #RB_Memórias.RB_Mem_Internas.RB_Prog_OK )
      S_Coil( #"RB.Di_PLC.Do"."RB.Di_PLC.Do17_ProgramaOK" )
   END_RUNG
   RUNG wire#w1
      I_Contact( #"RB.Do_PLC.Di"."RB.Do_PLC.Di17_RequisicaoPrograma" )
      R_Coil( #"RB.Di_PLC.Do"."RB.Di_PLC.Do17_ProgramaOK" )
   END_RUNG
   // the same network as SCL:
   IF #True AND #"RB.Do_PLC.Di"."RB.Do_PLC.Di17_RequisicaoPrograma" AND #RB_Memórias.RB_Mem_Internas.RB_Prog_OK THEN
       #"RB.Di_PLC.Do"."RB.Di_PLC.Do17_ProgramaOK" := TRUE;
   END_IF;
   IF #True AND NOT #"RB.Do_PLC.Di"."RB.Do_PLC.Di17_RequisicaoPrograma" THEN
       #"RB.Di_PLC.Do"."RB.Di_PLC.Do17_ProgramaOK" := FALSE;
   END_IF;
END_REGION

REGION Network 26: RB - Zera Numero de Programa
   RUNG wire#powerrail
      I_Contact( #"RB.Do_PLC.Di"."RB.Do_PLC.Di17_RequisicaoPrograma" )
      Contact( #RB_Memórias.RB_Mem_Internas.RB_Prog_OK )
      wire#w1
      Contact( #False )
      { S7_GenerateENO := "TRUE" } Move(in := INT#0, out1 => #"RB.Di_PLC.Do"."RB.Gi_PLC.Go_NumProg", out2 => #RB_Memórias.RB_Mem_Internas.RB_Mem_Prog_RB_Enviado)
   END_RUNG
   RUNG wire#powerrail
      Contact( #RB_Memórias.RB_Mem_Internas."Nenhuma Chamada Ativa" )
      { S7_Templates := "SrcType := Int" } NE_Contact(in1 := #RB_Memórias.RB_Mem_Internas.RB_Mem_Prog_RB_Enviado, in2 := 0)
   END_RUNG wire#w1
   // the same network as SCL:
   IF ((NOT #"RB.Do_PLC.Di"."RB.Do_PLC.Di17_RequisicaoPrograma" AND #RB_Memórias.RB_Mem_Internas.RB_Prog_OK) OR (#RB_Memórias.RB_Mem_Internas."Nenhuma Chamada Ativa" AND (#RB_Memórias.RB_Mem_Internas.RB_Mem_Prog_RB_Enviado <> 0))) AND #False THEN
       #"RB.Di_PLC.Do"."RB.Gi_PLC.Go_NumProg" := INT#0;
       #RB_Memórias.RB_Mem_Internas.RB_Mem_Prog_RB_Enviado := INT#0;
   END_IF;
END_REGION

REGION Network 27: #########################################
END_REGION

REGION Network 28: RB - CLP <-> Robo Anticolisao
END_REGION

NETWORK
TITLE = Salva
      LAR1  #SAVE_AR1;
      LAR2  #SAVE_AR2;
      SET;
      SAVE;
END_FUNCTION_BLOCK
